DATA_BLOCK "DB2035_PID"
TITLE = DB2035_PID
{ S7_Optimized_Access := 'FALSE' }
AUTHOR : AketzaBarragues
FAMILY : ZeusControl
VERSION : 1.0
//Bloque de datos dispositivo PID
   STRUCT
      PID { S7_SetPoint := 'False'} : Array[0.."N_MAX_DISP_PID"] of "UDT_ZC_DISP_PID";
      Mux { S7_SetPoint := 'False'} : Array[0.."N_MAX_MUX_DISP"] of "UDT_ZC_DISP_MUX_PID";
      Agrup : Array[0.."N_MAX_DISP_AGRUP"] of "UDT_ZC_DISP_AGRUP";
   END_STRUCT;


BEGIN
   PID[0].Estado_AutoMan := TRUE;
   PID[0].Estado_ModeActivate := FALSE;
   PID[0].Orden_Forzar := FALSE;
   PID[0].Orden_ActivarAuto := FALSE;
   PID[0].Orden_Ack := FALSE;
   PID[0].Orden_Reset := FALSE;
   PID[0].Alarmas_Error := FALSE;
   PID[0].Config_InvertirControl := FALSE;
   PID[0].Config_TipoEntrada := FALSE;
   PID[0].Aux_oldForzar := FALSE;
   PID[0].Estado_PV := 0.0;
   PID[0].Estado_ValorSalida := 0.0;
   PID[0].Estado_PV_0_100 := 0.0;
   PID[0].Estado_SP_0_100 := 0.0;
   PID[0].Estado_Error_SP_PV_0_100 := 0.0;
   PID[0].Estado_Mode := 3;
   PID[0].Estado_EstadoPID := 3;
   PID[0].Orden_ConsignaAuto := 0.0;
   PID[0].Orden_ConsignaForzado := 0.0;
   PID[0].Alarmas_ErrorBits := 16#0000_0000;
   PID[0].Config_Gain := 0.15;
   PID[0].Config_Ti := 3.0;
   PID[0].Config_Td := 0.0;
   PID[0].Config_LimiteSuperiorSalida := 100.0;
   PID[0].Config_LimiteInferiorSalida := 0.0;
   PID[0].Config_LimiteSuperiorEntrada := 15000.0;
   PID[0].Config_LimiteInferiorEntrada := 0.0;
   PID[0].Aux_oldMode := 3;
   PID[0].Aux_SP_Manual := 0.0;
   PID[0].Aux_SP_Auto := 0.0;
   PID[0].Aux_oldGain := 0.15;
   PID[0].Aux_oldTi := 3.0;
   PID[0].Aux_oldTd := 0.0;
   PID[1].Estado_AutoMan := TRUE;
   PID[1].Estado_ModeActivate := FALSE;
   PID[1].Orden_Forzar := FALSE;
   PID[1].Orden_ActivarAuto := FALSE;
   PID[1].Orden_Ack := FALSE;
   PID[1].Orden_Reset := FALSE;
   PID[1].Alarmas_Error := FALSE;
   PID[1].Config_InvertirControl := FALSE;
   PID[1].Config_TipoEntrada := FALSE;
   PID[1].Aux_oldForzar := FALSE;
   PID[1].Estado_PV := 1.085069;
   PID[1].Estado_ValorSalida := 0.0;
   PID[1].Estado_PV_0_100 := 0.003616898;
   PID[1].Estado_SP_0_100 := 0.0;
   PID[1].Estado_Error_SP_PV_0_100 := 0.003616898;
   PID[1].Estado_Mode := 4;
   PID[1].Estado_EstadoPID := 4;
   PID[1].Orden_ConsignaAuto := 0.0;
   PID[1].Orden_ConsignaForzado := 0.0;
   PID[1].Alarmas_ErrorBits := 16#0000_0000;
   PID[1].Config_Gain := 0.005;
   PID[1].Config_Ti := 8.0;
   PID[1].Config_Td := 0.0;
   PID[1].Config_LimiteSuperiorSalida := 100.0;
   PID[1].Config_LimiteInferiorSalida := 0.0;
   PID[1].Config_LimiteSuperiorEntrada := 30000.0;
   PID[1].Config_LimiteInferiorEntrada := 0.0;
   PID[1].Aux_oldMode := 4;
   PID[1].Aux_SP_Manual := 0.0;
   PID[1].Aux_SP_Auto := 0.0;
   PID[1].Aux_oldGain := 0.005;
   PID[1].Aux_oldTi := 8.0;
   PID[1].Aux_oldTd := 0.0;
   Mux[0].Habilitar := TRUE;
   Mux[0].ExisteCambio := FALSE;
   Mux[0].MaxVisible := FALSE;
   Mux[0].Index := 0;
   Mux[0].oldIndex := 0;
   Mux[0].PID.Estado_AutoMan := TRUE;
   Mux[0].PID.Estado_ModeActivate := FALSE;
   Mux[0].PID.Orden_Forzar := FALSE;
   Mux[0].PID.Orden_ActivarAuto := FALSE;
   Mux[0].PID.Orden_Ack := FALSE;
   Mux[0].PID.Orden_Reset := FALSE;
   Mux[0].PID.Alarmas_Error := FALSE;
   Mux[0].PID.Config_InvertirControl := FALSE;
   Mux[0].PID.Config_TipoEntrada := FALSE;
   Mux[0].PID.Aux_oldForzar := FALSE;
   Mux[0].PID.Estado_PV := 0.0;
   Mux[0].PID.Estado_ValorSalida := 0.0;
   Mux[0].PID.Estado_PV_0_100 := 0.0;
   Mux[0].PID.Estado_SP_0_100 := 0.0;
   Mux[0].PID.Estado_Error_SP_PV_0_100 := 0.0;
   Mux[0].PID.Estado_Mode := 3;
   Mux[0].PID.Estado_EstadoPID := 3;
   Mux[0].PID.Orden_ConsignaAuto := 0.0;
   Mux[0].PID.Orden_ConsignaForzado := 0.0;
   Mux[0].PID.Alarmas_ErrorBits := 16#0000_0000;
   Mux[0].PID.Config_Gain := 0.15;
   Mux[0].PID.Config_Ti := 3.0;
   Mux[0].PID.Config_Td := 0.0;
   Mux[0].PID.Config_LimiteSuperiorSalida := 100.0;
   Mux[0].PID.Config_LimiteInferiorSalida := 0.0;
   Mux[0].PID.Config_LimiteSuperiorEntrada := 15000.0;
   Mux[0].PID.Config_LimiteInferiorEntrada := 0.0;
   Mux[0].PID.Aux_oldMode := 3;
   Mux[0].PID.Aux_SP_Manual := 0.0;
   Mux[0].PID.Aux_SP_Auto := 0.0;
   Mux[0].PID.Aux_oldGain := 0.15;
   Mux[0].PID.Aux_oldTi := 3.0;
   Mux[0].PID.Aux_oldTd := 0.0;
   Mux[1].Habilitar := TRUE;
   Mux[1].ExisteCambio := FALSE;
   Mux[1].MaxVisible := FALSE;
   Mux[1].Index := 0;
   Mux[1].oldIndex := 0;
   Mux[1].PID.Estado_AutoMan := TRUE;
   Mux[1].PID.Estado_ModeActivate := FALSE;
   Mux[1].PID.Orden_Forzar := FALSE;
   Mux[1].PID.Orden_ActivarAuto := FALSE;
   Mux[1].PID.Orden_Ack := FALSE;
   Mux[1].PID.Orden_Reset := FALSE;
   Mux[1].PID.Alarmas_Error := FALSE;
   Mux[1].PID.Config_InvertirControl := FALSE;
   Mux[1].PID.Config_TipoEntrada := FALSE;
   Mux[1].PID.Aux_oldForzar := FALSE;
   Mux[1].PID.Estado_PV := 0.0;
   Mux[1].PID.Estado_ValorSalida := 0.0;
   Mux[1].PID.Estado_PV_0_100 := 0.0;
   Mux[1].PID.Estado_SP_0_100 := 0.0;
   Mux[1].PID.Estado_Error_SP_PV_0_100 := 0.0;
   Mux[1].PID.Estado_Mode := 3;
   Mux[1].PID.Estado_EstadoPID := 3;
   Mux[1].PID.Orden_ConsignaAuto := 0.0;
   Mux[1].PID.Orden_ConsignaForzado := 0.0;
   Mux[1].PID.Alarmas_ErrorBits := 16#0000_0000;
   Mux[1].PID.Config_Gain := 0.15;
   Mux[1].PID.Config_Ti := 3.0;
   Mux[1].PID.Config_Td := 0.0;
   Mux[1].PID.Config_LimiteSuperiorSalida := 100.0;
   Mux[1].PID.Config_LimiteInferiorSalida := 0.0;
   Mux[1].PID.Config_LimiteSuperiorEntrada := 15000.0;
   Mux[1].PID.Config_LimiteInferiorEntrada := 0.0;
   Mux[1].PID.Aux_oldMode := 3;
   Mux[1].PID.Aux_SP_Manual := 0.0;
   Mux[1].PID.Aux_SP_Auto := 0.0;
   Mux[1].PID.Aux_oldGain := 0.15;
   Mux[1].PID.Aux_oldTi := 3.0;
   Mux[1].PID.Aux_oldTd := 0.0;
   Agrup[0].AlgunaEnManual := TRUE;
   Agrup[0].AlgunaAlarma := FALSE;
   Agrup[0].NuevaAlarma := FALSE;
   Agrup[1].AlgunaEnManual := TRUE;
   Agrup[1].AlgunaAlarma := FALSE;
   Agrup[1].NuevaAlarma := FALSE;

END_DATA_BLOCK

